FUNCTION_BLOCK CoEResetTask EXTENDS MotionTask
VAR
	MCReset		  : MC_Reset;
	SequenceState : UDINT;
END_VAR

{attribute 'monitoring' := 'call'}
PROPERTY Busy : BOOL
GET
Busy := SequenceState <> 0;
END_GET
END_PROPERTY

METHOD CyclicLogic
CASE SequenceState OF
	0: // Wait for Execute()
	10:
		MCReset.Execute := TRUE;
		SequenceState	:= SequenceState + 10;

	20:
		IF NOT MCReset.Busy THEN
			SequenceState := 0;
		END_IF
END_CASE

MCReset(Axis := _Axis.Axis);
MCReset.Execute := FALSE;
END_METHOD

{attribute 'monitoring' := 'call'}
PROPERTY Error : BOOL
GET
Error := MCReset.Error;
END_GET
END_PROPERTY

{attribute 'monitoring' := 'call'}
PROPERTY ErrorId : UDINT
GET
ErrorId := MCReset.ErrorID;
END_GET
END_PROPERTY

METHOD Execute : BOOL
IF _Axis.Axis.Status.Coupled AND NOT _Axis.Axis.Status.Error THEN
	Execute := TRUE;
	RETURN;
ELSIF Busy OR _Axis.Axis.Status.Coupled THEN
	Execute := TRUE;
	RETURN;
END_IF

SequenceState := 10;
Execute		  := TRUE;
END_METHOD

END_FUNCTION_BLOCK

(* stored: Version 1.1.0.1, ProductVersion 3.1.4026.18
   POU CoEResetTask: Id {c0417bf1-f8e5-455c-b709-b1adca61b2e5}, SpecialFunc None
   Property Busy: Id {1756a8ef-6afd-4888-bbf5-c98a10bb54d0}
   Get Get: Id {36baa675-da67-4bbc-b138-3ed594a436e4}
   Method CyclicLogic: Id {372b78e9-314f-42e9-9970-18a442c41547}
   Property Error: Id {be55d477-4238-4c9d-b4bc-58e0cd557417}
   Get Get: Id {f06d8b23-37be-4526-b5cd-0cf3f263f6f9}
   Property ErrorId: Id {9e86757c-7ef1-4c06-8fb2-5fe5a8ef2101}
   Get Get: Id {a9f5a584-8a0b-4f20-a9a7-f96dde005a24}
   Method Execute: Id {98b589b7-73b6-40dd-bb4f-d1e78231dd89} *)
